(* CODESYS project Übung3.project

Project tree, tasks and I/O mapping:
  CODESYS_Control_Win_V3 : CODESYS Control Win V3, 3S - Smart Software Solutions GmbH, version 3.5.3.60
    application Application
      task VISU_TASK (cyclic, interval 100 ms, priority 30) calls VisuElems.Visu_Prg
      task Main_Task (cyclic, interval t#20ms, priority 1) calls Parkhaus
      program Parkhaus [LD]
      visualisation Parkhaus_Vis
  text list GlobalTextList
*)

// CODESYS_Control_Win_V3/Application/Parkhaus
PROGRAM Parkhaus
VAR
	M1: BOOL;
	LS1: BOOL;
	LS2: BOOL;
	Zaehler: INT := 0;
	Voll: BOOL;
	LS3: BOOL;
	M2: BOOL;
	LS4: BOOL;
	S1: BOOL;
	Reset: BOOL;
END_VAR
VAR // added by the converter: edge detectors and wires of the graphical bodies
    _w1, _w2, _w3 : BOOL;
END_VAR

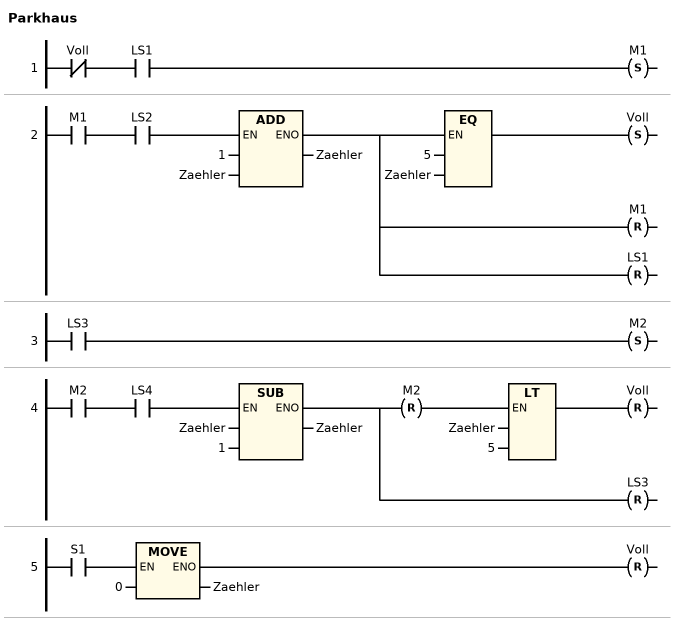
// NETWORK 1
M1 S= NOT Voll AND LS1;

// NETWORK 2
_w1 := M1 AND LS2;
IF _w1 THEN Zaehler := 1 + Zaehler; END_IF
Voll S= _w1 AND 5 = Zaehler;
M1 R= _w1;
LS1 R= _w1;

// NETWORK 3
M2 S= LS3;

// NETWORK 4
_w2 := M2 AND LS4;
IF _w2 THEN Zaehler := Zaehler - 1; END_IF
M2 R= _w2;
Voll R= _w2 AND Zaehler < 5;
LS3 R= _w2;

// NETWORK 5
_w3 := S1;
IF _w3 THEN Zaehler := 0; END_IF
Voll R= _w3;

END_PROGRAM

// CODESYS_Control_Win_V3/Application/Parkhaus_Vis
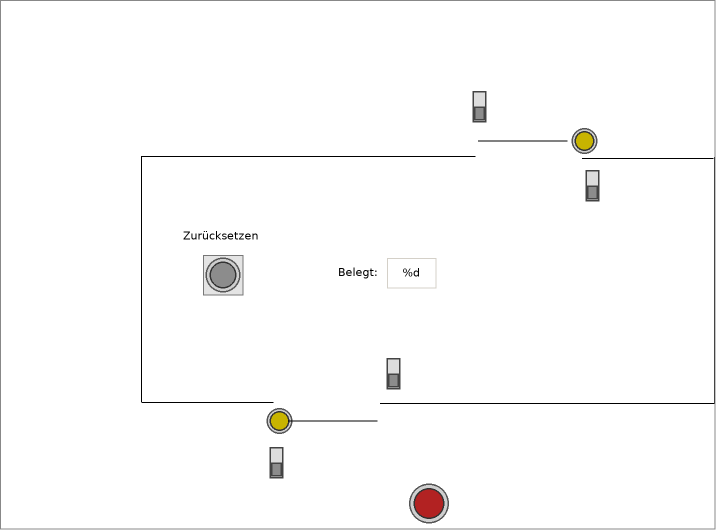
VISUALIZATION Parkhaus_Vis  // 716x530
    PushSwitch (202,255 42x40), tooltip "Zurücksetzen", variable: Parkhaus.S1, behaviour: TOGGLE, style: Switch-PushSwitch-Gray
    Label (173,221 96x30), "Zurücksetzen"
    Line (141,155)
    Line (141,156) (141,402)
    Line (142,402)
    Line (142,402) (273,402)
    Line (380,403) (714,403)
    Line (714,157) (714,403)
    Line (582,158) (713,158)
    Line (141,156) (475,156)
    Lamp1 (406,479 46x49), variable: Parkhaus.Voll, style: Lamp-Lamp1-Red
    Lamp1 (261,406 37x30), variable: Parkhaus.M1, style: Lamp-Lamp1-Yellow
    Lamp1 (566,126 37x30), variable: Parkhaus.M2, style: Lamp-Lamp1-Yellow
    Line (377,421) (288,421), invisible if: Parkhaus.M1
    Line (567,141) (478,141), invisible if: Parkhaus.M2
    Textfield (387,258 49x30), "%d", text variable: Parkhaus.Zaehler
    Label (329,259 58x27), "Belegt:"
    DipSwitch (260,447 33x31), tooltip "Lichtschranke 1", variable: Parkhaus.LS1, behaviour: TOGGLE, style: Switch-DipSwitch-Gray
    DipSwitch (377,358 33x31), tooltip "Lichtschranke 2", variable: Parkhaus.LS2, behaviour: TOGGLE, style: Switch-DipSwitch-Gray
    DipSwitch (576,170 33x31), tooltip "Lichtschranke 3", variable: Parkhaus.LS3, behaviour: TOGGLE, style: Switch-DipSwitch-Gray
    DipSwitch (463,91 33x31), tooltip "Lichtschranke 4", variable: Parkhaus.LS4, behaviour: TOGGLE, style: Switch-DipSwitch-Gray
END_VISUALIZATION
